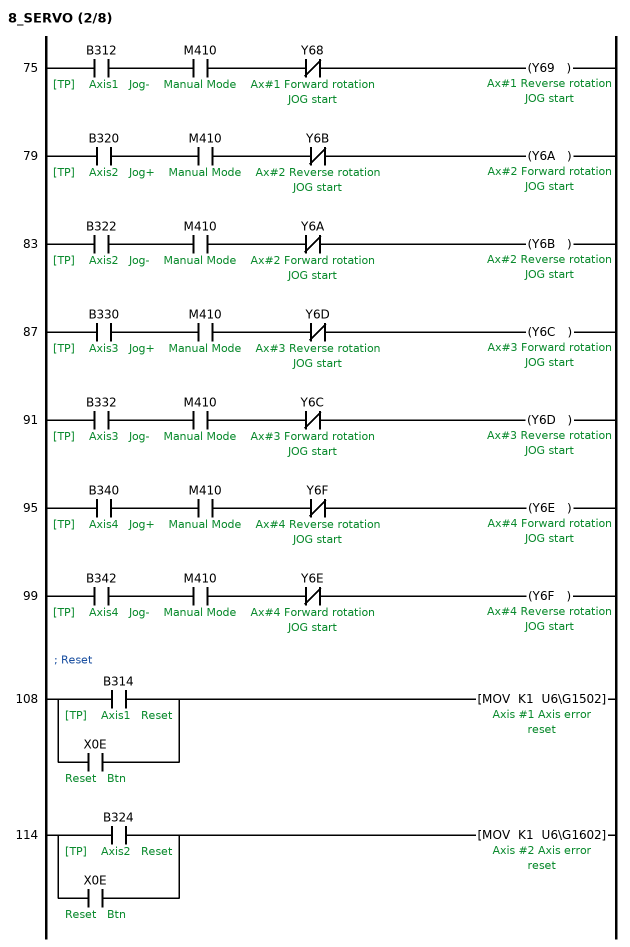
[picture p24: ladder of 8_SERVO, rungs at steps 75 to 114]
75    LD      B312  ; [TP]    Axis1   Jog-
      AND     M410  ; Manual Mode
      ANI     Y68  ; Ax#1 Forward rotation JOG start
      OUT     Y69  ; Ax#1 Reverse rotation JOG start
79    LD      B320  ; [TP]    Axis2   Jog+
      AND     M410  ; Manual Mode
      ANI     Y6B  ; Ax#2 Reverse rotation JOG start
      OUT     Y6A  ; Ax#2 Forward rotation JOG start
83    LD      B322  ; [TP]    Axis2   Jog-
      AND     M410  ; Manual Mode
      ANI     Y6A  ; Ax#2 Forward rotation JOG start
      OUT     Y6B  ; Ax#2 Reverse rotation JOG start
87    LD      B330  ; [TP]    Axis3   Jog+
      AND     M410  ; Manual Mode
      ANI     Y6D  ; Ax#3 Reverse rotation JOG start
      OUT     Y6C  ; Ax#3 Forward rotation JOG start
91    LD      B332  ; [TP]    Axis3   Jog-
      AND     M410  ; Manual Mode
      ANI     Y6C  ; Ax#3 Forward rotation JOG start
      OUT     Y6D  ; Ax#3 Reverse rotation JOG start
95    LD      B340  ; [TP]    Axis4   Jog+
      AND     M410  ; Manual Mode
      ANI     Y6F  ; Ax#4 Reverse rotation JOG start
      OUT     Y6E  ; Ax#4 Forward rotation JOG start
99    LD      B342  ; [TP]    Axis4   Jog-
      AND     M410  ; Manual Mode
      ANI     Y6E  ; Ax#4 Forward rotation JOG start
      OUT     Y6F  ; Ax#4 Reverse rotation JOG start
; Reset
108   LD      B314  ; [TP]    Axis1   Reset
      OR      X0E  ; Reset   Btn
      MOV     K1 U6\G1502  ; Axis #1 Axis error reset
114   LD      B324  ; [TP]    Axis2   Reset
      OR      X0E  ; Reset   Btn
      MOV     K1 U6\G1602  ; Axis #2 Axis error reset
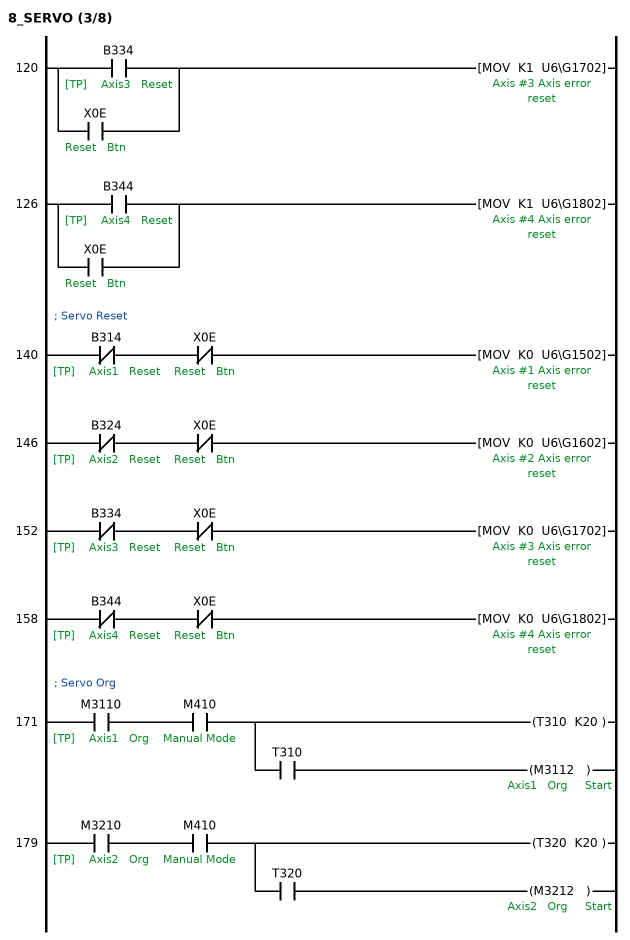
120   LD      B334  ; [TP]    Axis3   Reset
      OR      X0E  ; Reset   Btn
      MOV     K1 U6\G1702  ; Axis #3 Axis error reset
126   LD      B344  ; [TP]    Axis4   Reset
      OR      X0E  ; Reset   Btn
      MOV     K1 U6\G1802  ; Axis #4 Axis error reset
; Servo Reset
140   LDI     B314  ; [TP]    Axis1   Reset
      ANI     X0E  ; Reset   Btn
      MOV     K0 U6\G1502
146   LDI     B324  ; [TP]    Axis2   Reset
      ANI     X0E  ; Reset   Btn
      MOV     K0 U6\G1602
152   LDI     B334  ; [TP]    Axis3   Reset
      ANI     X0E  ; Reset   Btn
      MOV     K0 U6\G1702
158   LDI     B344  ; [TP]    Axis4   Reset
      ANI     X0E  ; Reset   Btn
      MOV     K0 U6\G1802
; Servo Org
171   LD      M3110  ; [TP]    Axis1   Org
      AND     M410  ; Manual Mode
      OUT     T310 K20
      AND     T310
      OUT     M3112  ; Axis1   Org     Start
179   LD      M3210  ; [TP]    Axis2   Org
      AND     M410  ; Manual Mode
      OUT     T320 K20
      AND     T320
      OUT     M3212  ; Axis2   Org     Start
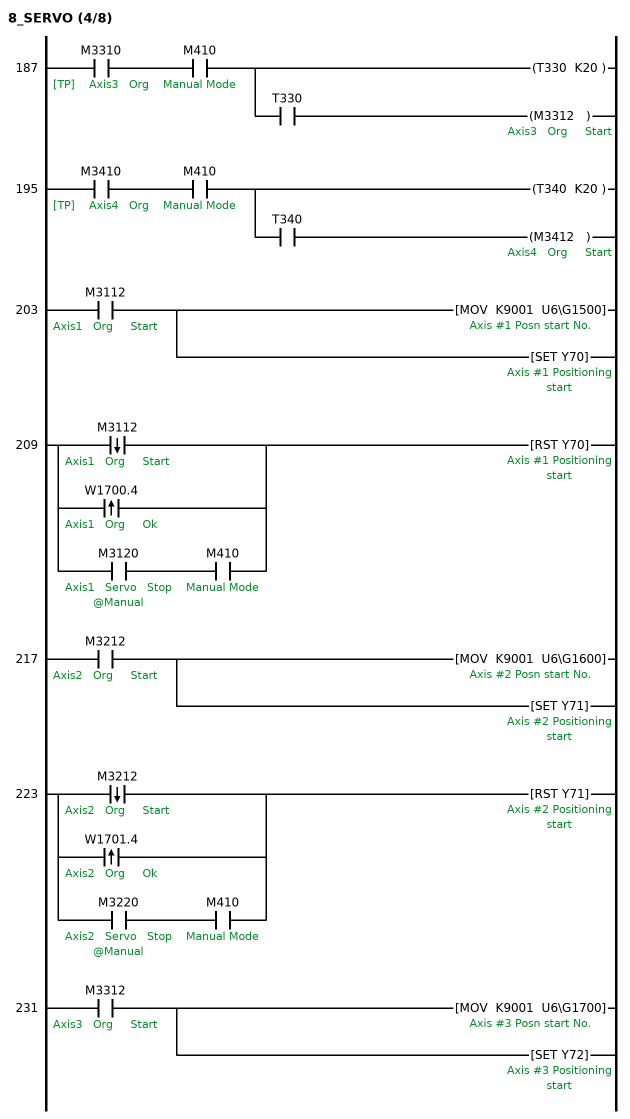
187   LD      M3310  ; [TP]    Axis3   Org
      AND     M410  ; Manual Mode
      OUT     T330 K20
      AND     T330
      OUT     M3312  ; Axis3   Org     Start
195   LD      M3410  ; [TP]    Axis4   Org
      AND     M410  ; Manual Mode
      OUT     T340 K20
      AND     T340
      OUT     M3412  ; Axis4   Org     Start
203   LD      M3112  ; Axis1   Org     Start
      MOV     K9001 U6\G1500  ; Axis #1 Posn start No.
      SET     Y70  ; Axis #1 Positioning start
209   LDF     M3112  ; Axis1   Org     Start
      ORP     W1700.4  ; Axis1   Org     Ok
      LD      M3120  ; Axis1   Servo   Stop    @Manual
      AND     M410  ; Manual Mode
      ORB
      RST     Y70  ; Axis #1 Positioning start
217   LD      M3212  ; Axis2   Org     Start
      MOV     K9001 U6\G1600  ; Axis #2 Posn start No.
      SET     Y71  ; Axis #2 Positioning start
223   LDF     M3212  ; Axis2   Org     Start
      ORP     W1701.4  ; Axis2   Org     Ok
      LD      M3220  ; Axis2   Servo   Stop    @Manual
      AND     M410  ; Manual Mode
      ORB
      RST     Y71  ; Axis #2 Positioning start
231   LD      M3312  ; Axis3   Org     Start
      MOV     K9001 U6\G1700  ; Axis #3 Posn start No.
      SET     Y72  ; Axis #3 Positioning start
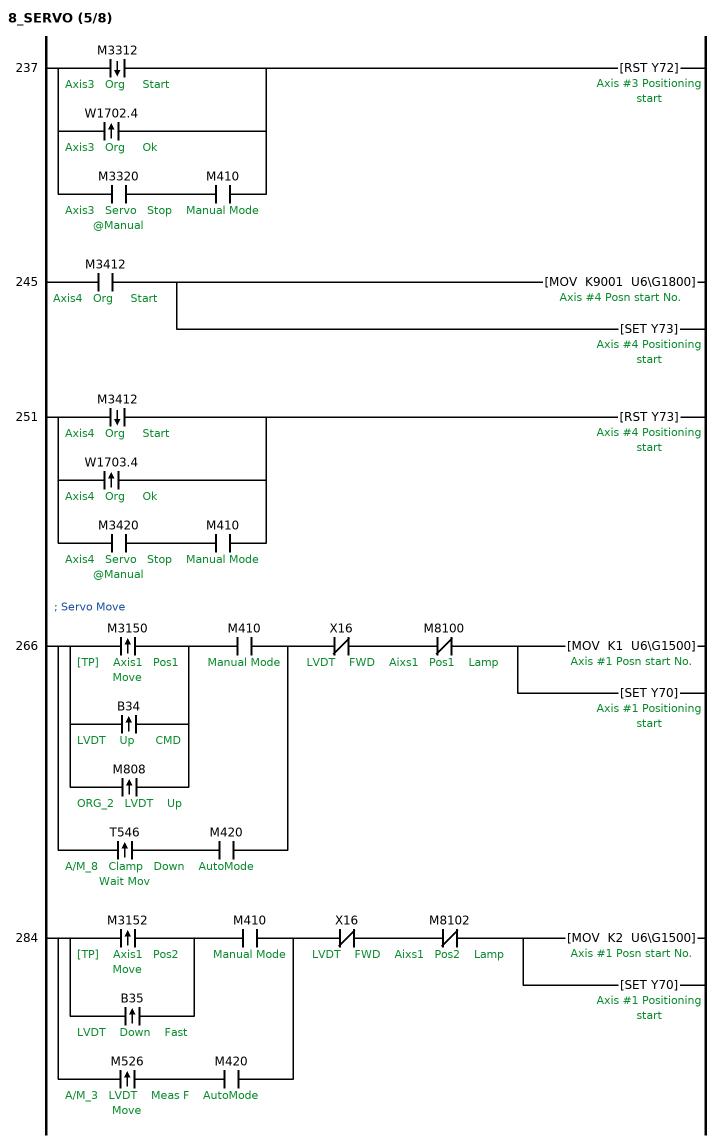
237   LDF     M3312  ; Axis3   Org     Start
      ORP     W1702.4  ; Axis3   Org     Ok
      LD      M3320  ; Axis3   Servo   Stop    @Manual
      AND     M410  ; Manual Mode
      ORB
      RST     Y72  ; Axis #3 Positioning start
245   LD      M3412  ; Axis4   Org     Start
      MOV     K9001 U6\G1800  ; Axis #4 Posn start No.
      SET     Y73  ; Axis #4 Positioning start
251   LDF     M3412  ; Axis4   Org     Start
      ORP     W1703.4  ; Axis4   Org     Ok
      LD      M3420  ; Axis4   Servo   Stop    @Manual
      AND     M410  ; Manual Mode
      ORB
      RST     Y73  ; Axis #4 Positioning start
; Servo Move
266   LDP     M3150  ; [TP]    Axis1   Pos1    Move
      ORP     B34  ; LVDT    Up      CMD
      ORP     M808  ; ORG_2   LVDT    Up
      AND     M410  ; Manual Mode
      LDP     T546  ; A/M_8   Clamp   Down    Wait Mov
      AND     M420  ; AutoMode
      ORB
      ANI     X16  ; LVDT    FWD
      ANI     M8100  ; Aixs1   Pos1    Lamp
      MOV     K1 U6\G1500
      SET     Y70  ; Axis #1 Positioning start
284   LDP     M3152  ; [TP]    Axis1   Pos2    Move
      ORP     B35  ; LVDT    Down    Fast
      AND     M410  ; Manual Mode
      LDP     M526  ; A/M_3   LVDT    Meas F  Move
      AND     M420  ; AutoMode
      ORB
      ANI     X16  ; LVDT    FWD
      ANI     M8102  ; Aixs1   Pos2    Lamp
      MOV     K2 U6\G1500
      SET     Y70  ; Axis #1 Positioning start
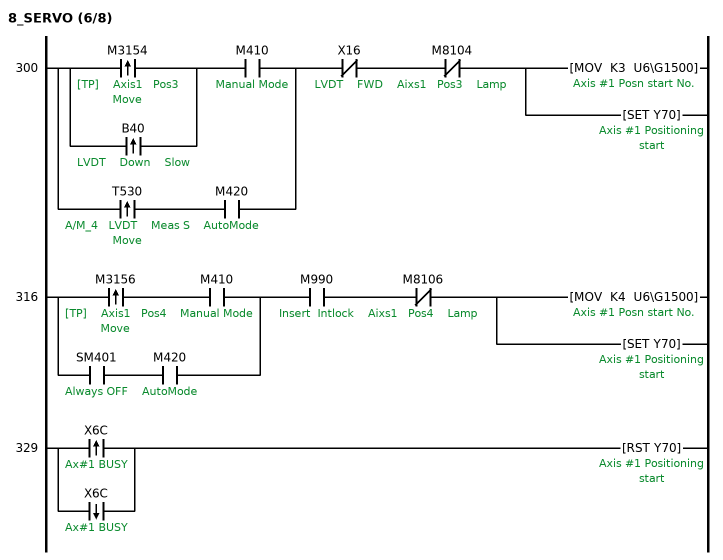
300   LDP     M3154  ; [TP]    Axis1   Pos3    Move
      ORP     B40  ; LVDT    Down    Slow
      AND     M410  ; Manual Mode
      LDP     T530  ; A/M_4   LVDT    Meas S  Move
      AND     M420  ; AutoMode
      ORB
      ANI     X16  ; LVDT    FWD
      ANI     M8104  ; Aixs1   Pos3    Lamp
      MOV     K3 U6\G1500
      SET     Y70  ; Axis #1 Positioning start
316   LDP     M3156  ; [TP]    Axis1   Pos4    Move
      AND     M410  ; Manual Mode
      LD      SM401  ; Always OFF
      AND     M420  ; AutoMode
      ORB
      AND     M990  ; Insert  Intlock
      ANI     M8106  ; Aixs1   Pos4    Lamp
      MOV     K4 U6\G1500
      SET     Y70  ; Axis #1 Positioning start
329   LDP     X6C  ; Ax#1 BUSY
      ORF     X6C  ; Ax#1 BUSY
      RST     Y70  ; Axis #1 Positioning start
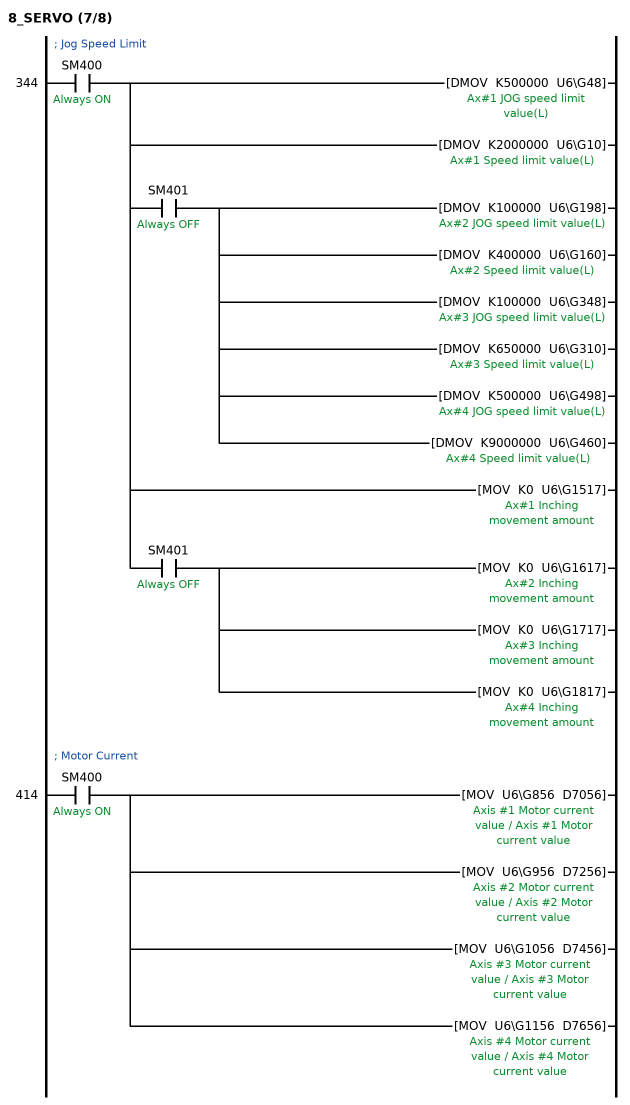
; Jog Speed Limit
344   LD      SM400  ; Always ON
      DMOV    K500000 U6\G48  ; Ax#1 JOG speed limit value(L)
      DMOV    K2000000 U6\G10  ; Ax#1 Speed limit value(L)
      MPS
      AND     SM401  ; Always OFF
      DMOV    K100000 U6\G198  ; Ax#2 JOG speed limit value(L)
      DMOV    K400000 U6\G160  ; Ax#2 Speed limit value(L)
      DMOV    K100000 U6\G348  ; Ax#3 JOG speed limit value(L)
      DMOV    K650000 U6\G310  ; Ax#3 Speed limit value(L)
      DMOV    K500000 U6\G498  ; Ax#4 JOG speed limit value(L)
      DMOV    K9000000 U6\G460  ; Ax#4 Speed limit value(L)
      MPP
      MOV     K0 U6\G1517  ; Ax#1 Inching movement amount
      AND     SM401  ; Always OFF
      MOV     K0 U6\G1617  ; Ax#2 Inching movement amount
      MOV     K0 U6\G1717  ; Ax#3 Inching movement amount
      MOV     K0 U6\G1817  ; Ax#4 Inching movement amount
; Motor Current
414   LD      SM400  ; Always ON
      MOV     U6\G856 D7056  ; Axis #1 Motor current value / Axis #1 Motor current value
      MOV     U6\G956 D7256  ; Axis #2 Motor current value / Axis #2 Motor current value
      MOV     U6\G1056 D7456  ; Axis #3 Motor current value / Axis #3 Motor current value
      MOV     U6\G1156 D7656  ; Axis #4 Motor current value / Axis #4 Motor current value
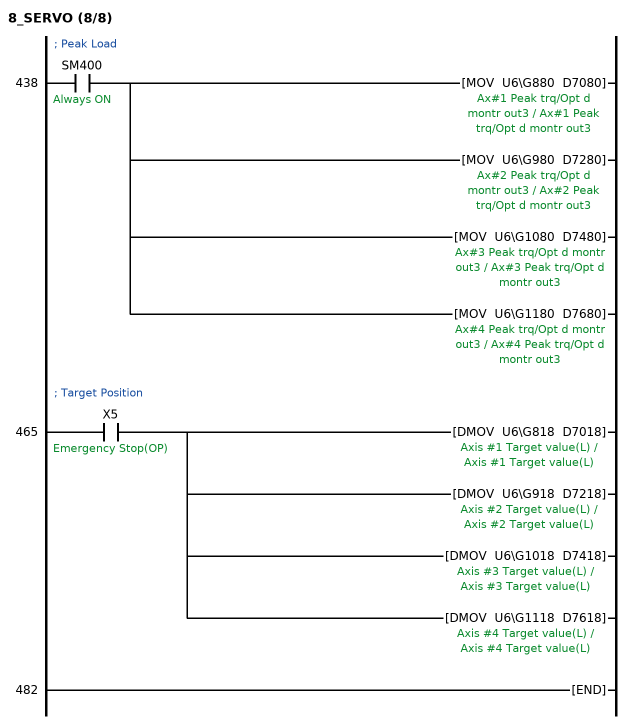
; Peak Load
438   LD      SM400  ; Always ON
      MOV     U6\G880 D7080  ; Ax#1 Peak trq/Opt d montr out3 / Ax#1 Peak trq/Opt d montr out3
      MOV     U6\G980 D7280  ; Ax#2 Peak trq/Opt d montr out3 / Ax#2 Peak trq/Opt d montr out3
      MOV     U6\G1080 D7480  ; Ax#3 Peak trq/Opt d montr out3 / Ax#3 Peak trq/Opt d montr out3
      MOV     U6\G1180 D7680  ; Ax#4 Peak trq/Opt d montr out3 / Ax#4 Peak trq/Opt d montr out3
; Target Position
465   LD      X5  ; Emergency Stop(OP)
      DMOV    U6\G818 D7018  ; Axis #1 Target value(L) / Axis #1 Target value(L)
      DMOV    U6\G918 D7218  ; Axis #2 Target value(L) / Axis #2 Target value(L)
      DMOV    U6\G1018 D7418  ; Axis #3 Target value(L) / Axis #3 Target value(L)
      DMOV    U6\G1118 D7618  ; Axis #4 Target value(L) / Axis #4 Target value(L)
482   END
END_PROGRAM

PROGRAM 9_MODEL
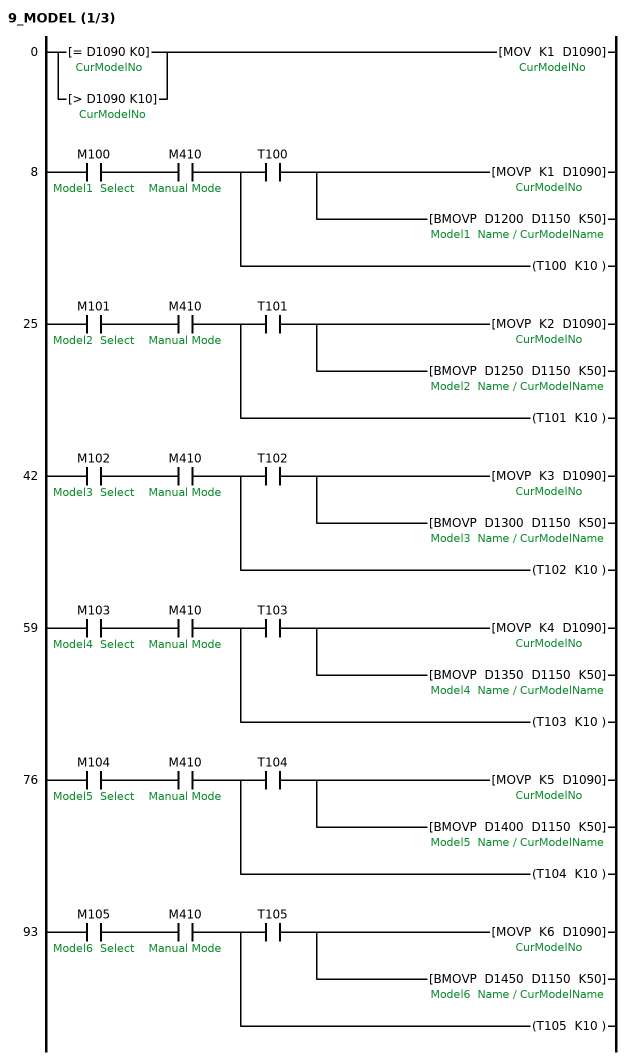
0     LD=     D1090 K0  ; CurModelNo
      OR>     D1090 K10  ; CurModelNo
      MOV     K1 D1090
8     LD      M100  ; Model1  Select
      AND     M410  ; Manual Mode
      MPS
      AND     T100
      MOVP    K1 D1090
      BMOVP   D1200 D1150 K50  ; Model1  Name / CurModelName
      MPP
      OUT     T100 K10
25    LD      M101  ; Model2  Select
      AND     M410  ; Manual Mode
      MPS
      AND     T101
      MOVP    K2 D1090
      BMOVP   D1250 D1150 K50  ; Model2  Name
      MPP
      OUT     T101 K10
42    LD      M102  ; Model3  Select
      AND     M410  ; Manual Mode
      MPS
      AND     T102
      MOVP    K3 D1090
      BMOVP   D1300 D1150 K50  ; Model3  Name
      MPP
      OUT     T102 K10
59    LD      M103  ; Model4  Select
      AND     M410  ; Manual Mode
      MPS
      AND     T103
      MOVP    K4 D1090
      BMOVP   D1350 D1150 K50  ; Model4  Name
      MPP
      OUT     T103 K10
76    LD      M104  ; Model5  Select
      AND     M410  ; Manual Mode
      MPS
      AND     T104
      MOVP    K5 D1090
      BMOVP   D1400 D1150 K50  ; Model5  Name
      MPP
      OUT     T104 K10
93    LD      M105  ; Model6  Select
      AND     M410  ; Manual Mode
      MPS
      AND     T105
      MOVP    K6 D1090
      BMOVP   D1450 D1150 K50  ; Model6  Name
      MPP
      OUT     T105 K10
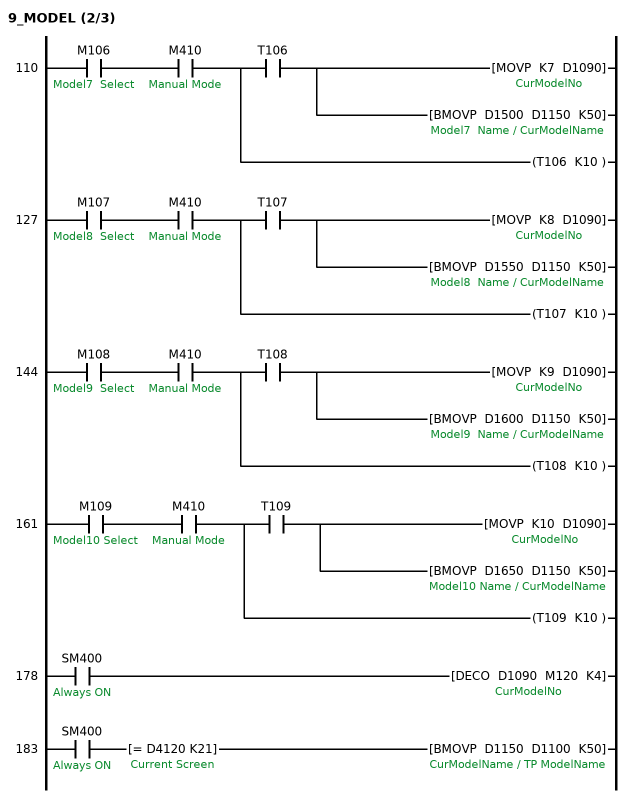
110   LD      M106  ; Model7  Select
      AND     M410  ; Manual Mode
      MPS
      AND     T106
      MOVP    K7 D1090
      BMOVP   D1500 D1150 K50  ; Model7  Name
      MPP
      OUT     T106 K10
127   LD      M107  ; Model8  Select
      AND     M410  ; Manual Mode
      MPS
      AND     T107
      MOVP    K8 D1090
      BMOVP   D1550 D1150 K50  ; Model8  Name
      MPP
      OUT     T107 K10
144   LD      M108  ; Model9  Select
      AND     M410  ; Manual Mode
      MPS
      AND     T108
      MOVP    K9 D1090
      BMOVP   D1600 D1150 K50  ; Model9  Name
      MPP
      OUT     T108 K10
161   LD      M109  ; Model10 Select
      AND     M410  ; Manual Mode
      MPS
      AND     T109
      MOVP    K10 D1090
      BMOVP   D1650 D1150 K50  ; Model10 Name
      MPP
      OUT     T109 K10
178   LD      SM400  ; Always ON
      DECO    D1090 M120 K4
183   LD      SM400  ; Always ON
      AND=    D4120 K21  ; Current Screen
      BMOVP   D1150 D1100 K50  ; TP ModelName
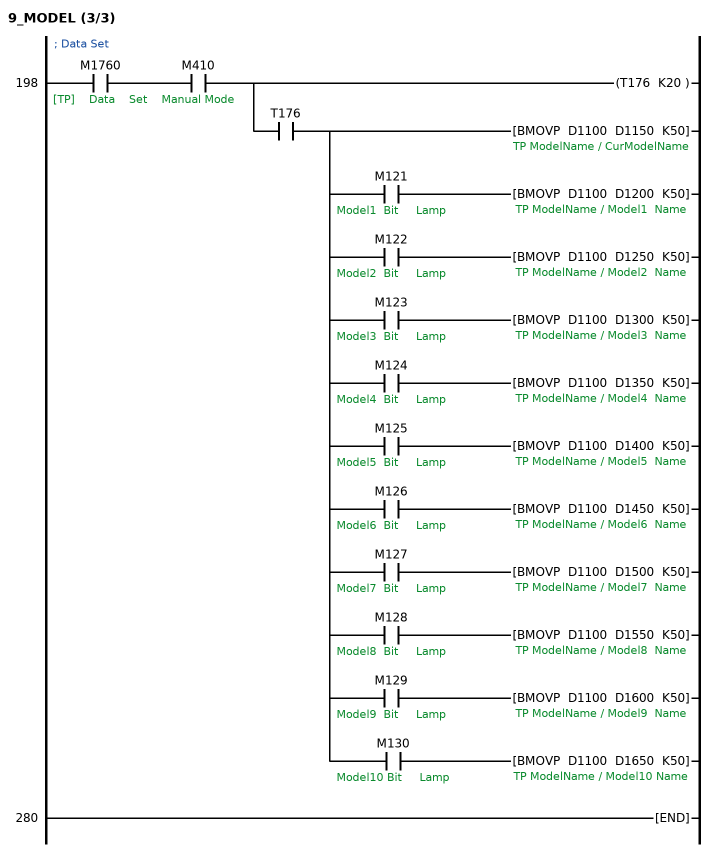
; Data Set
198   LD      M1760  ; [TP]    Data    Set
      AND     M410  ; Manual Mode
      OUT     T176 K20
      AND     T176
      BMOVP   D1100 D1150 K50
      MPS
      AND     M121  ; Model1  Bit     Lamp
      BMOVP   D1100 D1200 K50
      MRD
      AND     M122  ; Model2  Bit     Lamp
      BMOVP   D1100 D1250 K50
      MRD
      AND     M123  ; Model3  Bit     Lamp
      BMOVP   D1100 D1300 K50
      MRD
      AND     M124  ; Model4  Bit     Lamp
      BMOVP   D1100 D1350 K50
      MRD
      AND     M125  ; Model5  Bit     Lamp
      BMOVP   D1100 D1400 K50
      MRD
      AND     M126  ; Model6  Bit     Lamp
      BMOVP   D1100 D1450 K50
      MRD
      AND     M127  ; Model7  Bit     Lamp
      BMOVP   D1100 D1500 K50
      MRD
      AND     M128  ; Model8  Bit     Lamp
      BMOVP   D1100 D1550 K50
      MRD
      AND     M129  ; Model9  Bit     Lamp
      BMOVP   D1100 D1600 K50
      MPP
      AND     M130  ; Model10 Bit     Lamp
      BMOVP   D1100 D1650 K50
280   END
END_PROGRAM

// device comments not shown above
X0  ; Main    EMG     Stop
X0A  ; Indicator Running
X15  ; Lvdt down Sensor
X61  ; Synchronization flag
X64  ; Ax#1 M code ON
X65  ; Ax#2 M code ON
X66  ; Ax#3 M code ON
X67  ; Ax#4 M code ON
X68  ; Ax#1 Error detection
X69  ; Ax#2 Error detection
X6A  ; Ax#3 Error detection
X6B  ; Ax#4 Error detection
X6D  ; Ax#2 BUSY
X6E  ; Ax#3 BUSY
X6F  ; Ax#4 BUSY
X70  ; Ax#1 Start completed
X71  ; Ax#2 Start completed
X72  ; Ax#3 Start completed
X73  ; Ax#4 Start completed
X74  ; Ax#1 Positioning completed
X75  ; Ax#2 Positioning completed
X76  ; Ax#3 Positioning completed
X77  ; Ax#4 Positioning completed
Y2A  ; Servo 2 Power
Y2B  ; Servo 3 Power
Y2C  ; Servo 4 Power
Y74  ; Ax#1 Execution prohibition flag
Y75  ; Ax#2 Execution prohibition flag
Y76  ; Ax#3 Execution prohibition flag
Y77  ; Ax#4 Execution prohibition flag
B3D  ; Red Lamp
T500  ; A/M_4   INV Run Time
T535  ; A/M_5   Error
D750  ; Serial  Com'    Binary  Data
D1110  ; TP ModelZ-Axis  Pos1    Acc
D1112  ; TP ModelZ-Axis  Pos1    Dec
D1114  ; TP ModelZ-Axis  Pos1    Spd
D1116  ; TP ModelZ-Axis  Pos1    Pos
D1118  ; TP ModelZ-Axis  Pos2    Acc
D1120  ; TP ModelZ-Axis  Pos2    Dec
D1122  ; TP ModelZ-Axis  Pos2    Spd
D1124  ; TP ModelZ-Axis  Pos2    Pos
D1126  ; TP ModelZ-Axis  Pos3    Acc
D1128  ; TP ModelZ-Axis  Pos3    Dec
D1130  ; TP ModelZ-Axis  Pos3    Spd
D1132  ; TP ModelZ-Axis  Pos3    Pos
D1134  ; TP ModelZ-Axis  Pos4    Acc
D1136  ; TP ModelZ-Axis  Pos4    Dec
D1138  ; TP ModelZ-Axis  Pos4    Spd
D1140  ; TP ModelZ-Axis  Pos4    Pos
D1168  ; CurModelZ-Axis  Pos2    Acc
D1170  ; CurModelZ-Axis  Pos2    Dec
D1176  ; CurModelZ-Axis  Pos3    Acc
D1178  ; CurModelZ-Axis  Pos3    Dec
D1184  ; CurModelZ-Axis  Pos4    Acc
D1186  ; CurModelZ-Axis  Pos4    Dec
D1210  ; Model1  Z-Axis  Pos1    Acc
D1212  ; Model1  Z-Axis  Pos1    Dec
D1214  ; Model1  Z-Axis  Pos1    Spd
D1216  ; Model1  Z-Axis  Pos1    Pos
D1218  ; Model1  Z-Axis  Pos2    Acc
D1220  ; Model1  Z-Axis  Pos2    Dec
D1222  ; Model1  Z-Axis  Pos2    Spd
D1224  ; Model1  Z-Axis  Pos2    Pos
D1226  ; Model1  Z-Axis  Pos3    Acc
D1228  ; Model1  Z-Axis  Pos3    Dec
D1230  ; Model1  Z-Axis  Pos3    Spd
D1232  ; Model1  Z-Axis  Pos3    Pos
D1234  ; Model1  Z-Axis  Pos4    Acc
D1236  ; Model1  Z-Axis  Pos4    Dec
D1238  ; Model1  Z-Axis  Pos4    Spd
D1240  ; Model1  Z-Axis  Pos4    Pos
D1260  ; Model2  Z-Axis  Pos1    Acc
D1262  ; Model2  Z-Axis  Pos1    Dec
D1264  ; Model2  Z-Axis  Pos1    Spd
D1266  ; Model2  Z-Axis  Pos1    Pos
D1268  ; Model2  Z-Axis  Pos2    Acc
D1270  ; Model2  Z-Axis  Pos2    Dec
D1272  ; Model2  Z-Axis  Pos2    Spd
D1274  ; Model2  Z-Axis  Pos2    Pos
D1276  ; Model2  Z-Axis  Pos3    Acc
D1278  ; Model2  Z-Axis  Pos3    Dec
D1280  ; Model2  Z-Axis  Pos3    Spd
D1282  ; Model2  Z-Axis  Pos3    Pos
D1284  ; Model2  Z-Axis  Pos4    Acc
D1286  ; Model2  Z-Axis  Pos4    Dec
D1288  ; Model2  Z-Axis  Pos4    Spd
D1290  ; Model2  Z-Axis  Pos4    Pos
D1310  ; Model3  Z-Axis  Pos1    Acc
D1312  ; Model3  Z-Axis  Pos1    Dec
D1314  ; Model3  Z-Axis  Pos1    Spd
D1316  ; Model3  Z-Axis  Pos1    Pos
D1318  ; Model3  Z-Axis  Pos2    Acc
D1320  ; Model3  Z-Axis  Pos2    Dec
D1322  ; Model3  Z-Axis  Pos2    Spd
D1324  ; Model3  Z-Axis  Pos2    Pos
D1326  ; Model3  Z-Axis  Pos3    Acc
D1328  ; Model3  Z-Axis  Pos3    Dec
D1330  ; Model3  Z-Axis  Pos3    Spd
D1332  ; Model3  Z-Axis  Pos3    Pos
D1334  ; Model3  Z-Axis  Pos3    Acc
D1336  ; Model3  Z-Axis  Pos4    Dec
D1338  ; Model3  Z-Axis  Pos4    Spd
D1340  ; Model3  Z-Axis  Pos4    Pos
D1360  ; Model4  Z-Axis  Pos1    Acc
D1362  ; Model4  Z-Axis  Pos1    Dec
D1364  ; Model4  Z-Axis  Pos1    Spd
D1366  ; Model4  Z-Axis  Pos1    Pos
D1368  ; Model4  Z-Axis  Pos2    Acc
D1370  ; Model4  Z-Axis  Pos2    Dec
D1372  ; Model4  Z-Axis  Pos2    Spd
D1374  ; Model4  Z-Axis  Pos2    Pos
D1376  ; Model4  Z-Axis  Pos3    Acc
D1378  ; Model4  Z-Axis  Pos3    Dec
D1380  ; Model4  Z-Axis  Pos3    Spd
D1382  ; Model4  Z-Axis  Pos3    Pos
D1384  ; Model4  Z-Axis  Pos4    Acc
D1386  ; Model4  Z-Axis  Pos4    Dec
D1388  ; Model4  Z-Axis  Pos4    Spd
D1390  ; Model4  Z-Axis  Pos4    Pos
D1410  ; Model5  Z-Axis  Pos1    Acc
D1412  ; Model5  Z-Axis  Pos1    Dec
D1414  ; Model5  Z-Axis  Pos1    Spd
D1416  ; Model5  Z-Axis  Pos1    Pos
D1418  ; Model5  Z-Axis  Pos2    Acc
D1420  ; Model5  Z-Axis  Pos2    Dec
D1422  ; Model5  Z-Axis  Pos2    Spd
D1424  ; Model5  Z-Axis  Pos2    Pos
D1426  ; Model5  Z-Axis  Pos3    Acc
D1428  ; Model5  Z-Axis  Pos3    Dec
D1430  ; Model5  Z-Axis  Pos3    Spd
D1432  ; Model5  Z-Axis  Pos3    Pos
D1434  ; Model5  Z-Axis  Pos4    Acc
D1436  ; Model5  Z-Axis  Pos4    Dec
D1438  ; Model5  Z-Axis  Pos4    Spd
D1440  ; Model5  Z-Axis  Pos4    Pos
D1460  ; Model6  Z-Axis  Pos1    Acc
D1462  ; Model6  Z-Axis  Pos1    Dec
D1464  ; Model6  Z-Axis  Pos1    Spd
D1466  ; Model6  Z-Axis  Pos1    Pos
D1468  ; Model6  Z-Axis  Pos2    Acc
D1470  ; Model6  Z-Axis  Pos2    Dec
D1472  ; Model6  Z-Axis  Pos2    Spd
D1474  ; Model6  Z-Axis  Pos2    Pos
D1476  ; Model6  Z-Axis  Pos3    Acc
D1478  ; Model6  Z-Axis  Pos3    Dec
D1480  ; Model6  Z-Axis  Pos3    Spd
D1482  ; Model6  Z-Axis  Pos3    Pos
D1484  ; Model6  Z-Axis  Pos4    Acc
D1486  ; Model6  Z-Axis  Pos4    Dec
D1488  ; Model6  Z-Axis  Pos4    Spd
D1490  ; Model6  Z-Axis  Pos4    Pos
D1510  ; Model7  Z-Axis  Pos1    Acc
D1512  ; Model7  Z-Axis  Pos1    Dec
D1514  ; Model7  Z-Axis  Pos1    Spd
D1516  ; Model7  Z-Axis  Pos1    Pos
D1518  ; Model7  Z-Axis  Pos2    Acc
D1520  ; Model7  Z-Axis  Pos2    Dec
D1522  ; Model7  Z-Axis  Pos2    Spd
D1524  ; Model7  Z-Axis  Pos2    Pos
D1526  ; Model7  Z-Axis  Pos3    Acc
D1528  ; Model7  Z-Axis  Pos3    Dec
D1530  ; Model7  Z-Axis  Pos3    Spd
D1532  ; Model7  Z-Axis  Pos3    Pos
D1534  ; Model7  Z-Axis  Pos4    Acc
D1536  ; Model7  Z-Axis  Pos4    Dec
D1538  ; Model7  Z-Axis  Pos4    Spd
D1540  ; Model7  Z-Axis  Pos4    Pos
D1560  ; Model8  Z-Axis  Pos1    Acc
D1562  ; Model8  Z-Axis  Pos1    Dec
D1564  ; Model8  Z-Axis  Pos1    Spd
D1566  ; Model8  Z-Axis  Pos1    Pos
D1568  ; Model8  Z-Axis  Pos2    Acc
D1570  ; Model8  Z-Axis  Pos2    Dec
D1572  ; Model8  Z-Axis  Pos2    Spd
D1574  ; Model8  Z-Axis  Pos2    Pos
D1576  ; Model8  Z-Axis  Pos3    Acc
D1578  ; Model8  Z-Axis  Pos3    Dec
D1580  ; Model8  Z-Axis  Pos3    Spd
D1582  ; Model8  Z-Axis  Pos3    Pos
D1584  ; Model8  Z-Axis  Pos4    Acc
D1586  ; Model8  Z-Axis  Pos4    Dec
D1588  ; Model8  Z-Axis  Pos4    Spd
D1590  ; Model8  Z-Axis  Pos4    Pos
D1610  ; Model9  Z-Axis  Pos1    Acc
D1612  ; Model9  Z-Axis  Pos1    Dec
D1614  ; Model9  Z-Axis  Pos1    Spd
D1616  ; Model9  Z-Axis  Pos1    Pos
D1618  ; Model9  Z-Axis  Pos2    Acc
D1620  ; Model9  Z-Axis  Pos2    Dec
D1622  ; Model9  Z-Axis  Pos2    Spd
D1624  ; Model9  Z-Axis  Pos2    Pos
D1626  ; Model9  Z-Axis  Pos3    Acc
D1628  ; Model9  Z-Axis  Pos3    Dec
D1630  ; Model9  Z-Axis  Pos3    Spd
D1632  ; Model9  Z-Axis  Pos3    Pos
D1634  ; Model9  Z-Axis  Pos4    Acc
D1636  ; Model9  Z-Axis  Pos4    Dec
D1638  ; Model9  Z-Axis  Pos4    Spd
D1640  ; Model9  Z-Axis  Pos4    Pos
D1660  ; Model10 Z-Axis  Pos1    Acc
D1662  ; Model10 Z-Axis  Pos1    Dec
D1664  ; Model10 Z-Axis  Pos1    Spd
D1666  ; Model10 Z-Axis  Pos1    Pos
D1668  ; Model10 Z-Axis  Pos2    Acc
D1670  ; Model10 Z-Axis  Pos2    Dec
D1672  ; Model10 Z-Axis  Pos2    Spd
D1674  ; Model10 Z-Axis  Pos2    Pos
D1676  ; Model10 Z-Axis  Pos3    Acc
D1678  ; Model10 Z-Axis  Pos3    Dec
D1680  ; Model10 Z-Axis  Pos3    Spd
D1682  ; Model10 Z-Axis  Pos3    Pos
D1684  ; Model10 Z-Axis  Pos4    Acc
D1686  ; Model10 Z-Axis  Pos4    Dec
D1688  ; Model10 Z-Axis  Pos4    Spd
D1690  ; Model10 Z-Axis  Pos4    Pos
W1002  ; Axis2   Current Position
W1004  ; Axis3   Current Position
W1006  ; Axis4   Current Position
W1100  ; Axis1   Feedrate
W1102  ; Axis2   Feedrate
W1104  ; Axis3   Feedrate
W1106  ; Axis4   Feedrate
W1300  ; Axis1   Eff     Load
W1302  ; Axis2   Eff     Load
W1304  ; Axis3   Eff     Load
W1306  ; Axis4   Eff     Load
W1400  ; Axis1   Regen   Load    Ratio
W1401  ; Axis2   Regen   Load    Ratio
W1402  ; Axis3   Regen   Load    Ratio
W1403  ; Axis4   Regen   Load    Ratio
W1500  ; Axis1   Axis    Oper    Status
W1501  ; Axis2   Axis    Oper    Status
W1502  ; Axis3   Axis    Oper    Status
W1503  ; Axis4   Axis    Oper    Status
W1600  ; Axis1   Ext     Input   Sig
W1601  ; Axis2   Ext     Input   Sig
W1602  ; Axis3   Ext     Input   Sig
W1603  ; Axis4   Ext     Input   Sig
W1700  ; Axis1   Status
W1701  ; Axis2   Status
W1702  ; Axis3   Status
W1703  ; Axis4   Status
W1800  ; Axis1   Speed   Limit
W1802  ; Axis2   Speed   Limit
W1804  ; Axis3   Speed   Limit
W1806  ; Axis4   Speed   Limit
